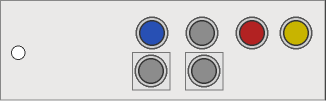
VISUALIZATION Control  // 326x101
VAR_IN_OUT
	LED_Blue : BOOL;
	LED_Red : BOOL;
	LED_White : BOOL;
	LED_Yellow : BOOL;
	Start : BOOL;
	Reset : BOOL;
	State : INT;
END_VAR
    Rectangle (0,0 326x100)
    Lamp1 (276,14 40x38), variable: LED_Yellow, style: Lamp-Lamp1-Yellow
    PushSwitch (182,52 44x38), variable: Start, behaviour: TAP, style: Switch-PushSwitch-Gray
    RadioButton (9,4 122x97), variable: State
        Areas[0]: Text=Off
        Areas[1]: Text=Manual
        Areas[2]: Text=Automatic
    Lamp1 (132,14 40x38), variable: LED_Blue, style: Lamp-Lamp1-Blue
    Lamp1 (232,14 40x38), variable: LED_Red, style: Lamp-Lamp1-Red
    Lamp1 (182,14 40x38), variable: LED_White, style: Lamp-Lamp1-Gray
    PushSwitch (129,52 44x38), variable: Reset, behaviour: TAP, style: Switch-PushSwitch-Gray
END_VISUALIZATION

(* stored: Version 1.1.0.1
   Visu Control: Id {74608ee7-0bed-4162-8008-406030be9e63} *)
